// TIA Portal V19 export
ORGANIZATION_BLOCK "OB1_ORCHESTRATOR"   // OB125, LAD, ProgramCycle
TITLE = "Main Program Sweep (Cycle)"
// stored: SetENOAutomatically false
   VAR_INPUT
      Initial_Call : Bool;   // Initial call of this OB
      Remanence : Bool;   // =True, if remanent data are available
   END_VAR
BEGIN

REGION Network 1
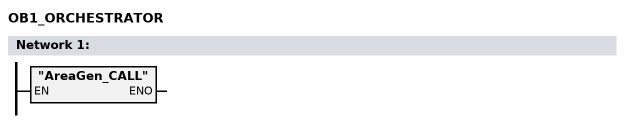
   RUNG wire#powerrail
      "AreaGen_CALL"()
   END_RUNG
   // the same network as SCL:
   "AreaGen_CALL"();
END_REGION
END_ORGANIZATION_BLOCK
